TYPE ST_WinchFeedback :
STRUCT
	length: LREAL;
	length_t: LREAL;
END_STRUCT
END_TYPE

(* stored: Version 1.1.0.1, ProductVersion 3.1.4022.7
   DUT ST_WinchFeedback: Id {e40b09e1-f0dd-4f61-8aff-a796c0bcc485} *)
